(* PLC project static_torsion.project, CODESYS CODESYS V3.5 SP17 Patch 3 *)
(* stored: creationDateTime 1970-01-01T00:00:00, modificationDateTime 2026-06-22T15:12:39.4699931 *)

TYPE PDI : STRUCT
  WDI : WORD;
  {attribute 'relative_offset' := '0'}
  CON_24V_ST : BIT;  (* 0 Питания +VES,+V04,+V05- в норме *)
  SAFE_A_ST : BIT;  (* 1 Реле безопасности #1 *)
  SAFE_B_ST : BIT;  (* 2 Реле безопасности #2 *)
  CON_220V_ST : BIT;  (* 3 Цепи управления 220V, вентиляция шкафа, вентиляторы на моторах *)
  UPS_24V_ST : BIT;  (* 4 Сигнал от ИБП - выходное напряжение ОК *)
  UPS_ACCU_BAD : BIT;  (* 5 Сигнал от ИБП - аккумулятор плохой *)
  UPS_ACCU_WORK : BIT;  (* 6 Сигнал от ИБП - работа от аккумулятора *)
  LS_UP : BIT;  (* 7 Аварийный КВ крайнее положение (Верх) *)
  LS_DN : BIT;  (* 8 Аварийный КВ крайнее положение (Низ) *)
  LS_BP : BIT;  (* 9 Снятие с концевика вертикальный силовозбудитель *)
  PWR_ST : BIT;  (* 10 Силовой контактор *)
  TRV_DRV_ACT : BIT;  (* 11 Привод подъёма траверсы активирован *)
  LS_DOOR : BIT;  (* 12 КВ "Дверь открыта" *)
  IN13 : BIT;  (* 13 *)
  IN14 : BIT;  (* 14 *)
  IN15 : BIT;  (* 15 *)
END_STRUCT;
END_TYPE
